// TIA Portal V21 export
TYPE "Std_Additivo"
   STRUCT
      In : Struct
         appo : Bool;
      END_STRUCT;
      Prm : Struct
         PercentualeAdditivoRich : Real;   // Percentuale di additivo richiesto
      END_STRUCT;
      Dati : Struct
         appo : Bool;
      END_STRUCT;
      Allarmi : Struct
         "A" : Array[0.."K_NumAllarmiPerAdditivi"] of "Std_PrmAllarmeStd";
         WordHMI : Word := 16#0000;
      END_STRUCT;
      Out : Struct
         AttualeAdditivo : Real;   // PortataAttualeTeorica(ql.i/h)
      END_STRUCT;
      Rif_Inc : Struct
         K_Analogica : Int;
         K_Motore : Int;
         K_Pid : Int;
      END_STRUCT;
   END_STRUCT;
END_TYPE
